FUNCTION_BLOCK SM_GForceMeasurement
VAR_INPUT
	///Measured raw milliG value (linked to I/O module)
	{attribute 'OPC.UA.DA' := '0'}
	milliGValue AT %I*: INT;
	///Error
	{attribute 'OPC.UA.DA' := '0'}
	error AT %I*: BOOL;
END_VAR
VAR_OUTPUT
	///Current status description
	{attribute 'OPC.UA.DA' := '1'}
	{attribute 'OPC.UA.DA.Access' := '1'}
	actualStatus: STRING;
	///Actual value
	{attribute 'OPC.UA.DA' := '1'}
	{attribute 'OPC.UA.DA.Access' := '1'}
	actual: GForce;
	///Moving average value
	{attribute 'OPC.UA.DA' := '1'}
	{attribute 'OPC.UA.DA.Access' := '1'}
	average: GForce;
	///Statuses of the state machine
	statuses: GForceMeasurementStatuses;
END_VAR
VAR_IN_OUT
END_VAR
VAR
END_VAR

actual( newMilliGValue := milliGValue );
statuses.healthStatus( isGood := NOT(error) );

END_FUNCTION_BLOCK

(* stored: Version 1.1.0.1, ProductVersion 3.1.4019.2
   POU SM_GForceMeasurement: Id {1dc586e1-5100-416e-934f-292342f88f08}, SpecialFunc None *)
